(* CoDeSys 2.3 export: ST_WB_VALVE_CFG.EXP *)

(* Data type *)
TYPE ST_WB_VALVE_CFG :
STRUCT
	Cycle   : REAL; (*Seconds*)
	TimeMax : REAL; (*Seconds*)
	PushTime: REAL; (*Seconds*)
	PushP   : REAL; (*Bar*)

	HP      : BYTE; (*Num. Pumps*)
END_STRUCT
END_TYPE
